// SIMATIC S7-200 project (STEP 7-Micro/WIN), CPU 222 REL 02.01

SYMBOL_TABLE ANWENDER1
SCHUTZSCHALTER   I0.7     // Motorschutzschalter
KREIS_1_STATUS   V0.0
KREIS_3_AUS      M1.0     // Kreis 3 ist ausgeschaltet.
KREIS_2_AUS      M0.7     // Kreis 2 ist ausgeschaltet.
KREIS_3_EIN      M0.6     // Kreis 3 ist angeschaltet.
KREIS_2_EIN      M0.5     // Kreis 2 ist angeschaltet.
ALARM_FILTER     M0.4     // Kein Wasser - Anlage abschalten!
ALARM_DRUCK      M0.3     // Druck zu niedrig - Kreis abschalten!
KEIN_DRUCK       I0.6     // Drucküberwachung im Kreis 1
FILTER           I0.5     // Drucküberwachung im Kreis 0.
PEGEL            M0.2     // Bodenfeucteregelung
BODEN_INT        VW92     // Potiwert Integer
BODEN_BYTE       SMB28    // Potiwert binär.
KREIS_1_OUT      Q0.1     // Kreis 1 Ausgang.
F4               V101.3   // Taste F4 von HMI
KREIS_1_AUS      M0.1     // Kreis 1 ist ausgeschaltet.
F1               V101.0   // Taste F1 von HMI
F2               V101.1   // Taste F2 von HMI
F3               V101.2   // Taste F3 von HMI.
KREIS_1_EIN      M0.0     // Kreis 1 ist angeschaltet.
END_SYMBOL_TABLE

ORGANIZATION_BLOCK MAIN:OB1
TITLE=PROGRAMMKOMMENTARE
BEGIN
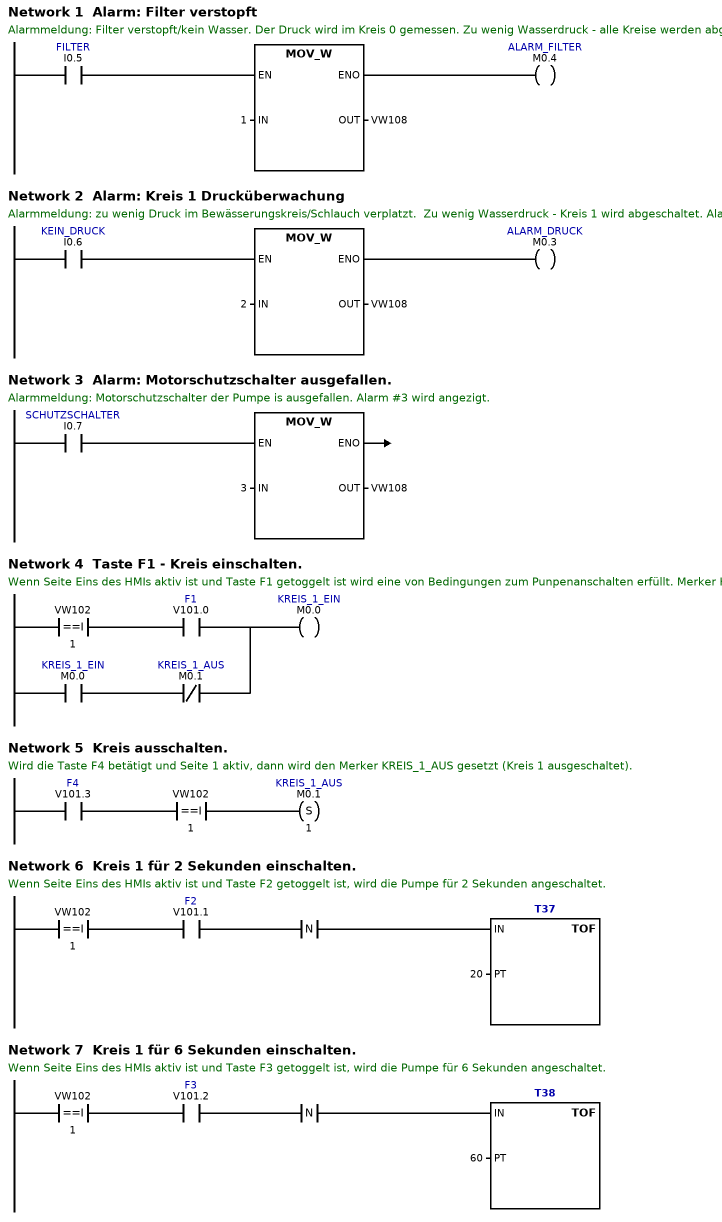
Network 1 // Alarm: Filter verstopft
// Alarmmeldung: Filter verstopft/kein Wasser. Der Druck wird im Kreis 0 gemessen. Zu wenig Wasserdruck - alle Kreise werden abgeschaltet. Alarm #1 wird aufgeblendet.
// (network saved uncompiled; LAD cells follow)
// row 0: c0 -| |- FILTER:I0.5  c1 --  c2 [MOV_W EN:=power@row0, IN:=1, ENO=>power, OUT=>VW108]  c3 --  c4 -( ) ALARM_FILTER:M0.4
// row 1: c2 [box]
Network 2 // Alarm: Kreis 1 Drucküberwachung
// Alarmmeldung: zu wenig Druck im Bewässerungskreis/Schlauch verplatzt.  Zu wenig Wasserdruck - Kreis 1 wird abgeschaltet. Alarm #2 wird aufgeblendet.
LD     KEIN_DRUCK:I0.6
MOVW   2, VW108
AENO
=      ALARM_DRUCK:M0.3
Network 3 // Alarm: Motorschutzschalter ausgefallen.
// Alarmmeldung: Motorschutzschalter der Pumpe is ausgefallen. Alarm #3 wird angezigt.
LD     SCHUTZSCHALTER:I0.7
MOVW   3, VW108
Network 4 // Taste F1 - Kreis einschalten.
// Wenn Seite Eins des HMIs aktiv ist und Taste F1 getoggelt ist wird eine von Bedingungen zum Punpenanschalten erfüllt. Merker KREIS_1_AUS schaltet die Bedingung KREIS_1_EIN ab.    
LDW=   VW102, 1
A      F1:V101.0
LD     KREIS_1_EIN:M0.0
AN     KREIS_1_AUS:M0.1
OLD
=      KREIS_1_EIN:M0.0
Network 5 // Kreis ausschalten.
// Wird die Taste F4 betätigt und Seite 1 aktiv, dann wird den Merker KREIS_1_AUS gesetzt (Kreis 1 ausgeschaltet).
LD     F4:V101.3
AW=    VW102, 1
S      KREIS_1_AUS:M0.1, 1
Network 6 // Kreis 1 für 2 Sekunden einschalten.
// Wenn Seite Eins des HMIs aktiv ist und Taste F2 getoggelt ist, wird die Pumpe für 2 Sekunden angeschaltet. 
// (network saved uncompiled; LAD cells follow)
// row 0: c0 -|==I|- VW102, 1  c1 -| |- F2:V101.1  c2 -|N|-  c3 --  c4 [TOF T37 IN:=power@row0, PT:=20]
// row 1: c4 [box]
Network 7 // Kreis 1 für 6 Sekunden einschalten.
// Wenn Seite Eins des HMIs aktiv ist und Taste F3 getoggelt ist, wird die Pumpe für 6 Sekunden angeschaltet. 
// (network saved uncompiled; LAD cells follow)
// row 0: c0 -|==I|- VW102, 1  c1 -| |- F3:V101.2  c2 -|N|-  c3 --  c4 [TOF T38 IN:=power@row0, PT:=60]
// row 1: c4 [box]
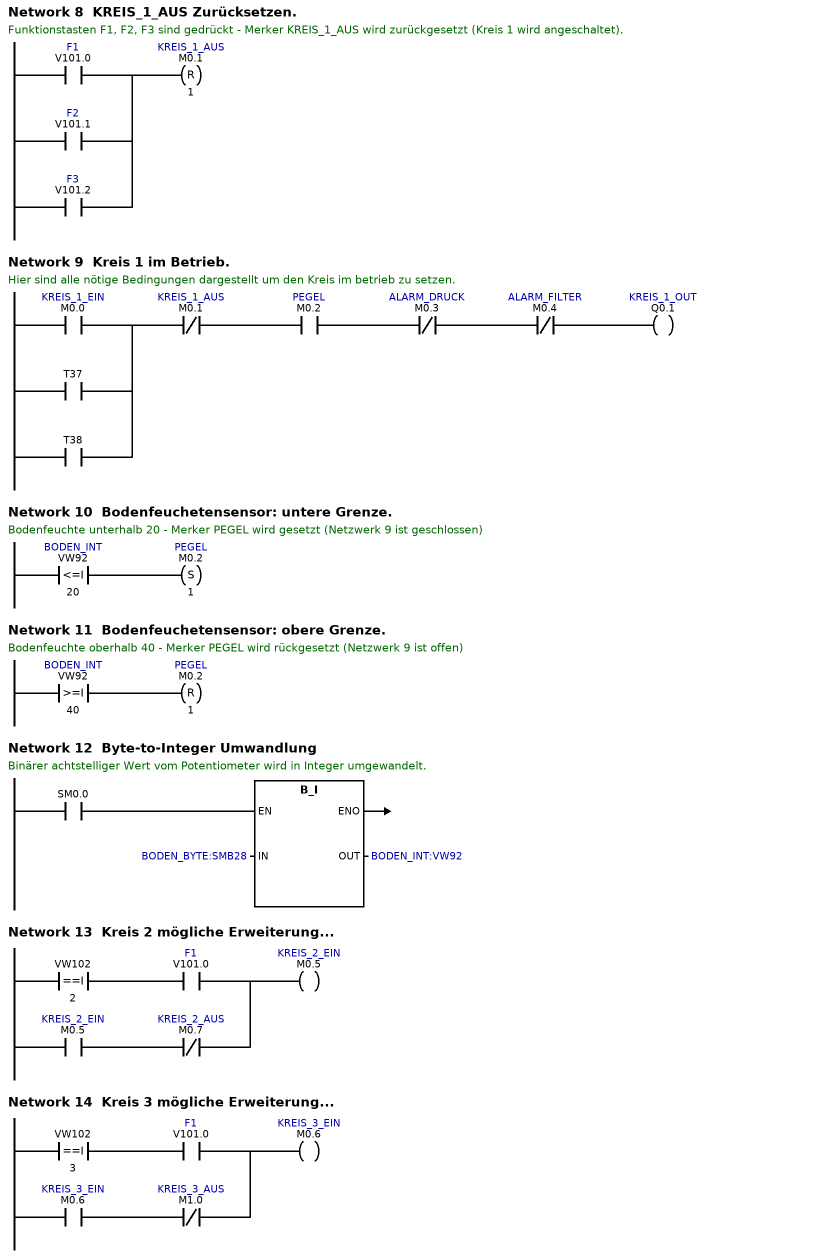
Network 8 // KREIS_1_AUS Zurücksetzen.
// Funktionstasten F1, F2, F3 sind gedrückt - Merker KREIS_1_AUS wird zurückgesetzt (Kreis 1 wird angeschaltet).
LD     F1:V101.0
O      F2:V101.1
O      F3:V101.2
R      KREIS_1_AUS:M0.1, 1
Network 9 // Kreis 1 im Betrieb.
// Hier sind alle nötige Bedingungen dargestellt um den Kreis im betrieb zu setzen.
LD     KREIS_1_EIN:M0.0
O      T37
O      T38
AN     KREIS_1_AUS:M0.1
A      PEGEL:M0.2
AN     ALARM_DRUCK:M0.3
AN     ALARM_FILTER:M0.4
=      KREIS_1_OUT:Q0.1
Network 10 // Bodenfeuchetensensor: untere Grenze.
// Bodenfeuchte unterhalb 20 - Merker PEGEL wird gesetzt (Netzwerk 9 ist geschlossen)
LDW<=  BODEN_INT:VW92, 20
S      PEGEL:M0.2, 1
Network 11 // Bodenfeuchetensensor: obere Grenze.
// Bodenfeuchte oberhalb 40 - Merker PEGEL wird rückgesetzt (Netzwerk 9 ist offen)
LDW>=  BODEN_INT:VW92, 40
R      PEGEL:M0.2, 1
Network 12 // Byte-to-Integer Umwandlung
// Binärer achtstelliger Wert vom Potentiometer wird in Integer umgewandelt.
LD     SM0.0
BTI    BODEN_BYTE:SMB28, BODEN_INT:VW92
Network 13 // Kreis 2 mögliche Erweiterung...
LDW=   VW102, 2
A      F1:V101.0
LD     KREIS_2_EIN:M0.5
AN     KREIS_2_AUS:M0.7
OLD
=      KREIS_2_EIN:M0.5
Network 14 // Kreis 3 mögliche Erweiterung...
LDW=   VW102, 3
A      F1:V101.0
LD     KREIS_3_EIN:M0.6
AN     KREIS_3_AUS:M1.0
OLD
=      KREIS_3_EIN:M0.6
END_ORGANIZATION_BLOCK
